PROGRAM MAIN
VAR
END_VAR

CalculatePrimeNumbers(10000);

END_PROGRAM

(* stored: Version 1.1.0.1, ProductVersion 3.1.4024.12
   POU MAIN: Id {375ad480-f07e-40c5-b818-4f06715483ed}, SpecialFunc None *)
